Universal Robots PolyScope program: move_to_base.urp

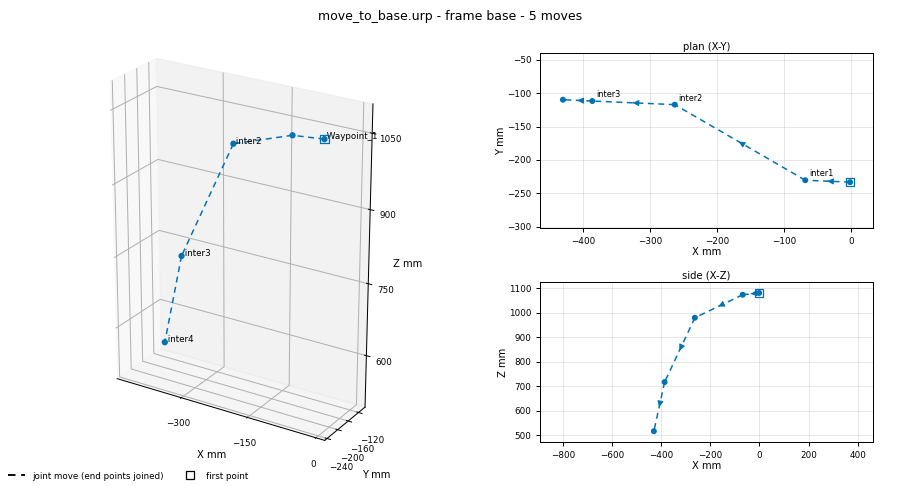
[picture p0: tool path of move_to_base.urp in frame base, 5 of 6 moves have a stored position in this frame; points joined in program order, loops and branches not executed]
Program move_to_base (installation=default directory=/programs/DND createdIn=5.12.4.1101661 lastSavedIn=5.12.4.1101661 robotSerialNumber=20225502378)
Calibrated DH parameters: a=[0.00022, -0.425328, -0.389701, 0.000059, 0.000065, 0]; d=[0.162608, 0.803456, 9.992211, -10.662202, 0.099702, 0.099559]; alpha=[1.570756, 0.001543, 0.004316, 1.570651, -1.570122, 0]; deltaTheta=[0, 0.002917, 0.116094, -0.119008, 0, -0.000001]
Robot Program (runOnlyOnce=true)
  MoveJ speed 60 deg/s, acceleration 80 deg/s^2 (useActiveTCP=true) feature=Base
    Waypoint Waypoint_1: TCP in base x=-1.285 y=-233.152 z=1080.057 mm, rx=-0.0065 ry=-2.2185 rz=2.2186 rad; joints [0.001, -89.999, 0.002, -89.999, 0.001, 0.001] deg
    Waypoint inter1: TCP in base x=-68.223 y=-230.306 z=1072.716 mm, rx=1.0931 ry=-1.343 rz=1.2867 rad; joints [-2.374, -92.35, 9.176, -80.518, -0.103, -97.404] deg
    Waypoint inter2: TCP in base x=-263.304 y=-117.317 z=978.94 mm, rx=0.0512 ry=-1.8258 rz=-0.172 rad; joints [-2.378, -100.858, 44.352, -108.971, -92.599, -97.761] deg
    Waypoint inter3: TCP in base x=-386.614 y=-111.884 z=716.74 mm, rx=0.1022 ry=-2.5843 rz=-0.1305 rad; joints [-2.376, -104.619, 78.203, -95.567, -92.628, -97.758] deg
    Waypoint inter4: TCP in base x=-430.462 y=-109.984 z=516.404 mm, rx=-0.1448 ry=3.1249 rz=0.0759 rad; joints [-2.389, -98.7, 93.692, -84.493, -92.599, -97.754] deg
    Waypoint Waypoint (Variable): variable=grid_base_hover
  URCap Gripper Activate (Robotiq_Grippers, Robotiq Inc.) dataModel(ResetAndActivateKey=false)
  URCap Gripper (Robotiq_Grippers, Robotiq Inc.) dataModel(position=75.0, force=0.0, speed=0.0, positionInDouble=75.0, forceInDouble=0.0, speedInDouble=0.0, slaveIds=[9], blocking=true)
